PROGRAM Simulation
VAR
	Lift1	:TON;
END_VAR

//Intake lift simulation:
IF HMI.stFromHMI.stLiftIntake.bGoUp THEN
	
	HMI.stFromHMI.stLiftIntake.bGoUp := FALSE;
END_IF

END_PROGRAM

(* stored: Version 1.1.0.1
   POU Simulation: Id {1c464058-24d6-42b5-95cd-ddd8975dc4d9}, SpecialFunc None *)
